{attribute 'qualified_only'}
VAR_GLOBAL
	// BT9 mirror
	temperature_mirror2		AT%I*: INT;
	// BT10
	temperature_mirror1		AT%I*: INT;

	//DOUT6 0.5
	brake_azimuth_eve	AT%Q*: BOOL;
	
	// DIN28 3.3 (absolute)
	azimut_limit_switch	AT%I*: BOOL;
	// DIN29 3.4
	focus_limit_near	AT%I*: BOOL;
	// DIN30 3.5
	focus_limit_far		AT%I*: BOOL;
	
	// DIN33 4.0
	cover1_open		AT%I*: BOOL;
	// DIN34 4.1
	cover1_closed	AT%I*: BOOL;
	// DIN35 4.2
	cover2_open		AT%I*: BOOL;
	// DIN36 4.3
	cover2_closed	AT%I*: BOOL;
	// DIN37 4.4
	cover3_open		AT%I*: BOOL;
	// DIN38 4.5
	cover3_closed	AT%I*: BOOL;

	//DOUT14 1.5
	focus_unlock		AT%Q*: BOOL;
	//Horn 4.7
	horn			AT%Q*: BOOL;
	
	// digitale inputs der Endlagen
	Derotator_inputs		AT%I*: WORD;
	// diagnostic number
	Derotator_diagnostic	AT%I*: UDINT;
	// derotator torque feedback
	Derotator_torque		AT%I*: INT;
	
	// digital inputs for limit switches
	Elevation_inputs		AT%I*: WORD;
	// diagnostic number
	Elevation_diagnostic	AT%I*: UDINT;
	// torque feedback
	Elevation_torque		AT%I*: INT;
	
	// digital inputs for limit switches
	Azimuth_inputs			AT%I*: WORD;
	// diagnostic number
	Azimuth_diagnostic		AT%I*: UDINT;
	// torque feedback
	Azimuth_torque			AT%I*: INT;
	
	// Zyklisches Interface zwischen NC und Achse
	AzimuthAxisRef: 	AXIS_REF;
	ElevationAxisRef: 	AXIS_REF;
	DerotatorAxisRef: 	AXIS_REF;
 	// Motor1 Channel 1
	FocusAxisRef:		AXIS_REF;
	
	//nasmyth_left	AT%Q*: BOOL;
	//nasmyth_right	AT%Q*: BOOL;
	open_cover1		AT%Q*: BOOL;
	close_cover1	AT%Q*: BOOL;
	open_cover2		AT%Q*: BOOL;
	close_cover2	AT%Q*: BOOL;
	open_cover3		AT%Q*: BOOL;
	close_cover3	AT%Q*: BOOL;
	
	
END_VAR

(* stored: Version 1.1.0.1, ProductVersion 3.1.4024.12
   GVL GVL_Telescope: Id {a7572ab9-17bf-4e0d-b71f-e76e531b6203} *)
